{attribute 'qualified_only'}
VAR_GLOBAL
	NUMBER_OF_SLOTS : INT := 6;
	SENSOR_POSITION_IN_DISC : INT := 4;
	
	// All the timeouts of the individual states are defined below as constants
	ROTATE_DISC_TIME: TIME := T#1S;
	LINEAR_FW_TIME: TIME := T#1500MS;
	GRIPPER_LOWER_TIME: TIME := T#1S;
	GRIPPER_OPEN_TIME: TIME := T#500MS;
	GRIPPER_CLOSE_TIME: TIME := T#500MS;
	GRIPPER_LIFT_TIME: TIME := T#1S;
	GRIPPER_LINEAR_BW_TIME: TIME := T#1500MS;
	
	TCP_SERVER_ADDRESS : STRING := '192.168.5.106';
	TCP_SERVER_PORT : UDINT := 9999;
	TOGGLE_BIT_TIME : TIME := T#500MS;
END_VAR

(* stored: Version 1.1.0.1, ProductVersion 3.1.4024.12
   GVL GVL: Id {3bb663e6-a027-427f-b62c-66381f90fed6} *)
